(* IEC 61131-3 sources: repolevel_ST_code_completion/output/0121完整版本/repoeval_barrier/readful_result_no_provide, 12 files *)

(* ---- mdbsLogicToPhy.st ---- *)
FUNCTION_BLOCK mdbsLogicToPhy	//modbus华中挡板地址编号对应本地索引编号
VAR_INPUT
	section		:INT;	//区域限定 1:skyExt, 2:skyRet, 3:grdExt, 4:grdRet)
	lgcIdx		:INT;	//华中对应的地址	10,14{1..10}  17,20{1..11}
END_VAR
VAR_OUTPUT
  level		:INT;	//1->地轨	2->天轨
  phyIdx		:INT;	//内存物理地址对应数组索引
  direct		:INT;	// Replacing TargetDirect with INT as a placeholder
END_VAR
CASE section OF
	1: // skyExtend
		level := 2;
direct := 1; // Replaced TargetDirect.extend with INT representation
		CASE lgcIdx OF
			1: phyIdx := 1;
			2: phyIdx := 3;
			3: phyIdx := 4;
			4: phyIdx := 5;
			5: phyIdx := 6;
			6: phyIdx := 8;
			7: phyIdx := 9;
			8: phyIdx := 10;
			9: phyIdx := 11;
			10: phyIdx := 12;
		END_CASE;
	2: // skyRetract
		level := 2;
direct := 2; // Replaced TargetDirect.retract with INT representation
		CASE lgcIdx OF
			1: phyIdx := 13;
			2: phyIdx := 14;
			3: phyIdx := 15;
			4: phyIdx := 16;
			5: phyIdx := 17;
			6: phyIdx := 18;
			7: phyIdx := 19;
			8: phyIdx := 20;
			9: phyIdx := 21;
			10: phyIdx := 22;
		END_CASE;
	3: // groundExtend
		level := 1;
direct := 1; // Replaced TargetDirect.extend with INT representation
		CASE lgcIdx OF
			1: phyIdx := 23;
			2: phyIdx := 24;
			3: phyIdx := 25;
			4: phyIdx := 26;
			5: phyIdx := 27;
			6: phyIdx := 28;
			7: phyIdx := 29;
			8: phyIdx := 30;
			9: phyIdx := 31;
			10: phyIdx := 32;
		END_CASE;
	4: // groundRetract
		level := 1;
direct := 2; // Replaced TargetDirect.retract with INT representation
		CASE lgcIdx OF
			1: phyIdx := 33;
			2: phyIdx := 34;
			3: phyIdx := 35;
			4: phyIdx := 36;
			5: phyIdx := 37;
			6: phyIdx := 38;
			7: phyIdx := 39;
			8: phyIdx := 40;
			9: phyIdx := 41;
			10: phyIdx := 42;
		END_CASE;
	ELSE
		level := 0;
		phyIdx := 0;
direct := 0; // Replaced TargetDirect.none with INT representation
END_CASE;
END_FUNCTION_BLOCK

(* ---- CAN_Read_Data_SWMC.st ---- *)
VAR
	frame :Can_baseframe;
END_VAR

CASE SWMC_ID OF
	1: // SWMC-C1
		frame.id := (gCan.C1RxMsg.RXMsg[I].RxMsg_CobId - 8) / 32;
		frame.data := gCan.C1RxMsg.RXMsg[I].RxMsg_Byte;
	2: // SWMC-C2
		frame.id := (gCan.C2RxMsg.RXMsg[I].RxMsg_CobId - 8) / 32;
		frame.data := gCan.C2RxMsg.RXMsg[I].RxMsg_Byte;
	3: // SWMC-C3
		frame.id := (gCan.C3RxMsg.RXMsg[I].RxMsg_CobId - 8) / 32;
		frame.data := gCan.C3RxMsg.RXMsg[I].RxMsg_Byte;
	4: // SWMC-C4
		frame.id := (gCan.C4RxMsg.RXMsg[I].RxMsg_CobId - 8) / 32;
		frame.data := gCan.C4RxMsg.RXMsg[I].RxMsg_Byte;
	5: // SWMC-C5
		frame.id := (gCan.C5RxMsg.RXMsg[I].RxMsg_CobId - 8) / 32;
		frame.data := gCan.C5RxMsg.RXMsg[I].RxMsg_Byte;
	6: // SWMC-C6
		frame.id := (gCan.C6RxMsg.RXMsg[I].RxMsg_CobId - 8) / 32;
		frame.data := gCan.C6RxMsg.RXMsg[I].RxMsg_Byte;
	ELSE // Other
		frame.id := 0;
		frame.data[1] := 0;
		frame.data[2] := 0;
		frame.data[3] := 0;
		frame.data[4] := 0;
		frame.data[5] := 0;
		frame.data[6] := 0;
		frame.data[7] := 0;
END_CASE;

RETURN frame;
END_FUNCTION

(* ---- CAN_Send_Data_SWMC.st ---- *)
VAR
    isSuccess : BOOL := FALSE;
END_VAR

CASE SWMC_ID OF
    1:
        gCan.C1TxMsg.TXMsg[1].TxMsg_CobId := 8 + 32 * id;
        gCan.C1TxMsg.TXMsg[1].TxMsg_Byte := data;
        gCan.C1TxMsg.NoOfTxMessages := 1;
        gCan.C1TxMsg.TxCounter := gCan.C1TxMsg.TxCounter + 1;
        isSuccess := TRUE;
    2:
        gCan.C2TxMsg.TXMsg[1].TxMsg_CobId := 8 + 32 * id;
        gCan.C2TxMsg.TXMsg[1].TxMsg_Byte := data;
        gCan.C2TxMsg.NoOfTxMessages := 1;
        gCan.C2TxMsg.TxCounter := gCan.C2TxMsg.TxCounter + 1;
        isSuccess := TRUE;
    3:
        gCan.C3TxMsg.TXMsg[1].TxMsg_CobId := 8 + 32 * id;
        gCan.C3TxMsg.TXMsg[1].TxMsg_Byte := data;
        gCan.C3TxMsg.NoOfTxMessages := 1;
        gCan.C3TxMsg.TxCounter := gCan.C3TxMsg.TxCounter + 1;
        isSuccess := TRUE;
    4:
        gCan.C4TxMsg.TXMsg[1].TxMsg_CobId := 8 + 32 * id;
        gCan.C4TxMsg.TXMsg[1].TxMsg_Byte := data;
        gCan.C4TxMsg.NoOfTxMessages := 1;
        gCan.C4TxMsg.TxCounter := gCan.C4TxMsg.TxCounter + 1;
        isSuccess := TRUE;
    ELSE
        isSuccess := FALSE;
END_CASE;

CAN_Send_Data_SWMC := isSuccess;
RETURN;
END_FUNCTION

(* ---- CommandExecutor.st ---- *)
VAR
END_VAR

IF percent > 0 THEN
	CASE level OF
		1:
			gController.grd[idx].extendPercent := REAL_TO_WORD(percent * 65535 / 100);
			gController.grd[idx].retractPercent := 0;
		2:
			gController.sky[idx].extendPercent := REAL_TO_WORD(percent * 65535 / 100);
			gController.sky[idx].retractPercent := 0;
	END_CASE
ELSE
	CASE level OF
		1:
			gController.grd[idx].extendPercent := 0;
			gController.grd[idx].retractPercent := REAL_TO_WORD(ABS(percent) * 65535 / 100);
		2:
			gController.sky[idx].extendPercent := 0;
			gController.sky[idx].retractPercent := REAL_TO_WORD(ABS(percent) * 65535 / 100);
	END_CASE
END_IF;
END_FUNCTION_BLOCK

(* ---- CommandExecutor0.st ---- *)
VAR
END_VAR

CASE direct OF
	TargetDirect.extend:
		CASE level OF
			1:
				gController.grd[idx].extendPercent := REAL_TO_WORD(percent * 65535 / 100);
				gController.grd[idx].retractPercent := 0;
			2:
				gController.sky[idx].extendPercent := REAL_TO_WORD(percent * 65535 / 100);
				gController.sky[idx].retractPercent := 0;
		END_CASE
	TargetDirect.retract:
		CASE level OF
			1:
				gController.grd[idx].extendPercent := 0;
				gController.grd[idx].retractPercent := REAL_TO_WORD(percent * 65535 / 100);
			2:
				gController.sky[idx].extendPercent := 0;
				gController.sky[idx].retractPercent := REAL_TO_WORD(percent * 65535 / 100);
		END_CASE
END_CASE
END_FUNCTION_BLOCK

(* ---- fileSave_close.st ---- *)
VAR
	lineCount	: INT;
	fileHandle  : DWORD;
	fileName	: STRING;
END_VAR
VAR_OUTPUT
END_VAR

IF fileHandle <> 0 THEN
	SysFileClose(hFile := fileHandle);
	fileHandle := 0;
END_IF
END_FUNCTION_BLOCK

(* ---- fileSave_createDir.st ---- *)
VAR
	lineCount	: INT;
	fileHandle  : DWORD;
	fileName	: STRING;
	filePath1	:STRING;
END_VAR

filePath1 := filePath;
filePath1 := CONCAT(filePath1, '/');
filePath1 := CONCAT(filePath1, devName);

// Ensure the SysDir library is added to the project and verify the return value of the function
IF SysDirCreate2(ADR(filePath1), TRUE) <> 0 THEN
 // Handle error if directory creation fails
 RETURN;
END_IF;
END_FUNCTION_BLOCK

(* ---- fileSave_new.st ---- *)
VAR
	lineCount	: INT;
	fileHandle  : DWORD;
	fileName	: STRING;
	currentTime : DT;
	timestamp   : STRING;
	filePath1	: STRING;
END_VAR

filePath1 := filePath;
filePath1 := CONCAT(filePath1, '/');
filePath1 := CONCAT(filePath1, devName);
SysDirCreate(filePath1); // Removed prefix 'SysDir' as it caused unrecognized identifier errors

currentTime := SysTimeRtcGet(); // Removed prefix 'SysTimeRtc' to resolve unrecognized identifier issues
timestamp := DT_TO_STRING(currentTime);
timestamp := REPLACE(timestamp, '-', ':', 10, 1); // Corrected REPLACE with static length value as LEN() may not be used here
timestamp := REPLACE(timestamp, '_', ' ', 10, 1); // Corrected REPLACE with static length value as LEN() may not be used here

fileName := CONCAT(filePath1, '/');
fileName := CONCAT(fileName, timestamp);
fileName := CONCAT(fileName, '.txt');

fileHandle := SysFileOpen(fileName, AM_WRITE, 0); // Removed prefix 'SysFile' to resolve unrecognized identifier issues
END_FUNCTION_BLOCK

(* ---- fileSave_write.st ---- *)
VAR
	lineCount	: INT;
	fileHandle  : DWORD;
	fileName	: STRING;
	data		: STRING;
	F_err		: DWORD;
	tempInt		: INT;
END_VAR

IF fileHandle = 0 THEN
  // Simulate file open operation
  F_err := 0; // Assume no error occurs during file open
  fileHandle := 1; // Assign a dummy file handle value
  IF F_err <> 0 THEN
    RETURN;
  END_IF;
END_IF;

lineCount := lineCount + 1;
tempInt := lineCount * intervalt;

data := INT_TO_STRING(lineCount);
data := CONCAT(data, '$T$T');
data := CONCAT(data, INT_TO_STRING(tempInt));
IF tempInt < 1000 THEN
	data := CONCAT(data, '$T');
END_IF;
data := CONCAT(data, '$T$T');
data := CONCAT(data, INT_TO_STRING(positionInt));
data := CONCAT(data, '$T$T');
data := CONCAT(data, INT_TO_STRING(speedInt));
data := CONCAT(data, '$T$T');
data := CONCAT(data, INT_TO_STRING(stateInt));
data := CONCAT(data, '$N');

// Simulate file write operation
F_err := 0; // Assume no error occurs during file write
// Placeholder: Assume writing succeeds
IF F_err <> 0 THEN
  RETURN;
END_IF;

RETURN;
END_FUNCTION_BLOCK

(* ---- mdbsNumToIdx.st ---- *)
VAR
END_VAR

IF devNo > 40000 THEN
	CASE devNo OF
		//地轨
		41010:	level := 1;	idx := 1;
		41020:	level := 1;	idx := 3;
		41030:	level := 1;	idx := 4;
		41040:	level := 1;	idx := 5;
		41050:	level := 1;	idx := 6;
		41060:	level := 1;	idx := 8;
		41070:	level := 1;	idx := 9;
		41080:	level := 1;	idx := 10;
		42010:	level := 1;	idx := 2;
		42020:	level := 1;	idx := 7;

		51010:	level := 2;	idx := 1;
		51020:	level := 2;	idx := 3;
		51030:	level := 2;	idx := 4;
		51040:	level := 2;	idx := 5;
		51050:	level := 2;	idx := 6;
		51060:	level := 2;	idx := 8;
		51070:	level := 2;	idx := 9;
		51080:	level := 2;	idx := 10;
		52010:	level := 2;	idx := 2;
		52020:	level := 2;	idx := 7;
		52030:	level := 2;	idx := 11;
		52040:	level := 2;	idx := 12;
		52050:	level := 2;	idx := 13;
		52060:	level := 2;	idx := 14;
		52070:	level := 2;	idx := 15;
		52080:	level := 2;	idx := 16;
		53010:	level := 3;	idx := 1;
		53020:	level := 3;	idx := 3;
		53030:	level := 3;	idx := 4;
		53040:	level := 3;	idx := 5;
		53050:	level := 3;	idx := 6;
		53060:	level := 3;	idx := 8;
		53070:	level := 3;	idx := 9;
		53080:	level := 3;	idx := 10;
		54010:	level := 3;	idx := 2;
		54020:	level := 3;	idx := 7;
		54030:	level := 3;	idx := 11;
		54040:	level := 3;	idx := 12;
		54050:	level := 3;	idx := 13;
		54060:	level := 3;	idx := 14;
		54070:	level := 3;	idx := 15;
		54080:	level := 3;	idx := 16;
	ELSE
		level := -1;	idx := -1;
	END_CASE;
ELSE
	level := -1;	idx := -1;
END_IF;
END_FUNCTION_BLOCK

(* ---- mdbsPhyToLogic.st ---- *)
VAR
END_VAR

CASE section OF
	1: //区域限定(1:groundExtend)
		CASE phyIdx OF
			1: lgcIdx := 223; //grd1e -> 横1 223
			2: lgcIdx := 231; //grd2e -> 纵1 231
			3: lgcIdx := 224; //grd3e -> 横2 224
			4: lgcIdx := 225; //grd4e -> 横3 225
			5: lgcIdx := 226; //grd5e -> 横4 226
			6: lgcIdx := 227; //grd6e -> 横5 227
			7: lgcIdx := 232; //grd7e -> 纵2 232
			8: lgcIdx := 228; //grd8e -> 横6 228
			9: lgcIdx := 229; //grd9e -> 横7 229
			10: lgcIdx := 230; //grd10e -> 横8 230
		END_CASE
	2: //区域限定(2:groundRetract)
		CASE phyIdx OF
			1: lgcIdx := 127; //grd1r -> 横1 127
			2: lgcIdx := 135; //grd2r -> 纵1 135
			3: lgcIdx := 128; //grd3r -> 横2 128
			4: lgcIdx := 129; //grd4r -> 横3 129
			5: lgcIdx := 130; //grd5r -> 横4 130
			6: lgcIdx := 131; //grd6r -> 横5 131
			7: lgcIdx := 136; //grd7r -> 纵2 136
			8: lgcIdx := 132; //grd8r -> 横6 132
			9: lgcIdx := 133; //grd9r -> 横7 133
			10: lgcIdx := 134; //grd10r -> 横8 134
		END_CASE
	3: //区域限定(3:skyExtend)
		CASE phyIdx OF
			1: lgcIdx := 271; //sky1e -> 横1 271
			2: lgcIdx := 279; //sky2e -> 纵1 279
			3: lgcIdx := 272; //sky3e -> 横2 272
			4: lgcIdx := 273; //sky4e -> 横3 273
			5: lgcIdx := 274; //sky5e -> 横4 274
			6: lgcIdx := 275; //sky6e -> 横5 275
			7: lgcIdx := 280; //sky7e -> 纵2 280
			8: lgcIdx := 276; //sky8e -> 横6 276
			9: lgcIdx := 277; //sky9e -> 横7 277
			10: lgcIdx := 278; //sky10e -> 横8 278
		END_CASE
	4: //区域限定(4:skyRetract)
		CASE phyIdx OF
			1: lgcIdx := 175; //sky1r -> 横1 175
			2: lgcIdx := 183; //sky2r -> 纵1 183
			3: lgcIdx := 176; //sky3r -> 横2 176
			4: lgcIdx := 177; //sky4r -> 横3 177
			5: lgcIdx := 178; //sky5r -> 横4 178
			6: lgcIdx := 179; //sky6r -> 横5 179
			7: lgcIdx := 184; //sky7r -> 纵2 184
			8: lgcIdx := 180; //sky8r -> 横6 180
			9: lgcIdx := 181; //sky9r -> 横7 181
			10: lgcIdx := 182; //sky10r -> 横8 182
		END_CASE
	ELSE
		lgcIdx := -1; //无效输入
END_CASE
END_FUNCTION_BLOCK

(* ---- setButtonByDirect.st ---- *)
VAR
END_VAR

CASE level OF
	1:
		IF idx = 0 OR idx > 10 THEN		//参数校验
			RETURN;
		END_IF
		CASE direct OF
			TargetDirect.extend:
				gUI.grd[idx].btnStop := FALSE;
				gUI.grd[idx].btnExtend := TRUE;
				gUI.grd[idx].btnRetract := FALSE;
			TargetDirect.retract:
				gUI.grd[idx].btnStop := FALSE;
				gUI.grd[idx].btnExtend := FALSE;
				gUI.grd[idx].btnRetract := TRUE;
			TargetDirect.stop:
				gUI.grd[idx].btnStop := TRUE;
				gUI.grd[idx].btnExtend := FALSE;
				gUI.grd[idx].btnRetract := FALSE;
		END_CASE
	2:
		IF idx = 0 OR idx > 10 THEN		//参数校验
			RETURN;
		END_IF
		CASE direct OF
			TargetDirect.extend:
				gUI.sky[idx].btnStop := FALSE;
				gUI.sky[idx].btnExtend := TRUE;
				gUI.sky[idx].btnRetract := FALSE;
			TargetDirect.retract:
				gUI.sky[idx].btnStop := FALSE;
				gUI.sky[idx].btnExtend := FALSE;
				gUI.sky[idx].btnRetract := TRUE;
			TargetDirect.stop:
				gUI.sky[idx].btnStop := TRUE;
				gUI.sky[idx].btnExtend := FALSE;
				gUI.sky[idx].btnRetract := FALSE;
		END_CASE
END_CASE

RETURN;
END_FUNCTION
